// TwinCAT 3 PLC project Main
// ProgramVersion: 3.1.4023.0
// libraries:
//   Tc2_Standard, * (Beckhoff Automation GmbH)
//   Tc2_System, * (Beckhoff Automation GmbH)
//   Tc3_Module, * (Beckhoff Automation GmbH)
// project tree:
//   DUTs/ Controller.TcDUT
//   GVLs/ Global.TcGVL
//   / PlcTask.TcTTO
//   POUs/ MAIN.TcPOU
// real-time tasks:
//   TASK PlcTask: cycle T#10ms, priority 20, ADS port 350

CONFIGURATION Main
    RESOURCE PLC ON TwinCAT3
        TASK PlcTask(INTERVAL := T#10ms, PRIORITY := 20);
        PROGRAM MAIN WITH PlcTask : MAIN;
    END_RESOURCE
END_CONFIGURATION

// ---- DUTs/Controller.TcDUT
TYPE Controller :
STRUCT
	LeftJoystickX : INT;
	LeftJoystickY : INT;
	RightJoystickX : INT;
	RightJoystickY : INT;
	LeftTrigger : INT;
	RightTrigger : INT;
	LeftBumper : BOOL;
	RightBumper : BOOL;
	ButtonA : BOOL;
	ButtonB : BOOL;
	ButtonX : BOOL;
	ButtonY : BOOL;
	LeftThumb : BOOL;
	RightThumb : BOOL;
	Back : BOOL;
	Start : BOOL;
	DPadX : INT;
	DPadY : INT;
END_STRUCT
END_TYPE

// ---- GVLs/Global.TcGVL
{attribute 'qualified_only'}
VAR_GLOBAL
	controller : Controller;
END_VAR

// ---- POUs/MAIN.TcPOU
PROGRAM MAIN
VAR
END_VAR

END_PROGRAM
